Yaskawa INFORM job: R1_W03,5,7(0,0)OK-KM.JBI

/JOB
//NAME R1_W03,5,7(0,0)OK-KM
///FOLDERNAME KRIS-SCIANA
//POS
///NPOS 94,94,0,4,0,0
///TOOL 0
///POSTYPE PULSE
///PULSE
C00000=-97801,-92951,-68020,-42573,91743,12282
C00001=-188064,-59139,-49719,-51220,48350,5801
C00002=-182482,-29523,-13831,-58220,47542,10694
C00003=-186503,-14327,-833,-57181,45005,9773
C00004=-186887,-13436,-157,-57022,44797,9650
C00005=-187358,-18276,-5525,-56185,44980,9089
C00006=-193250,-27913,-6363,-58294,38967,9969
C00007=-199995,-16364,1412,-54222,35645,7165
C00008=-199327,-15584,1994,-54497,36056,7364
C00009=-199882,-17213,782,-54333,35681,7234
C00010=-195511,-15034,9725,-61255,35872,11434
C00011=-195511,-14418,11078,-61887,35615,11785
C00012=-194782,-15937,9357,-61766,36202,11793
C00013=-185148,-27392,-13403,-56780,46393,9588
C00014=-194611,-49573,-33459,-572,31924,22077
C00015=-195793,-42632,-27790,753,32004,21336
C00016=-196651,-38308,-23003,1749,31294,20781
C00017=-197052,-37261,-22343,2197,31434,20529
C00018=-196235,-39864,-25459,1248,31997,21059
C00019=-202582,-39238,-15691,30047,22851,6468
C00020=-202582,-38747,-14553,30589,22461,6206
C00021=-199520,-48265,-22642,26019,21519,8620
C00022=-195597,-45769,-34616,-8656,41829,26358
C00023=-205752,-37498,-18561,12983,36783,12907
C00024=-204602,-36516,-17940,11961,36728,13544
C00025=-195976,-39153,-18531,-9623,35365,26897
C00026=-197793,-59286,-35313,-7977,35152,25873
C00027=-213331,-48054,-41686,-15165,61809,-3623
C00028=-205738,-19523,-29471,-74829,71236,-32232
C00029=-213283,8162,-7439,-90948,66894,-41154
C00030=-215606,11272,-4686,-90700,65214,-41123
C00031=-216577,12559,-3127,-90719,64506,-40980
C00032=-216866,14771,-1122,-90727,64291,-40934
C00033=-216575,12516,-3571,-90601,64514,-41108
C00034=-216096,11995,12560,-96030,67022,-42309
C00035=-217024,11210,11856,-96058,66343,-42301
C00036=-218189,6682,-8739,-75138,67073,-44258
C00037=-217766,7327,-6835,-75554,67132,-43814
C00038=-218002,9228,-4372,-75728,66817,-43579
C00039=-221147,-8168,-21082,-78731,52920,-40929
C00040=-218126,-14316,-25848,-79593,55000,-40534
C00041=-213331,-48054,-41686,-15165,61809,-3623
C00042=-211970,-37779,-14430,-6801,34223,-17849
C00043=-210033,-36470,-13605,-8545,34568,-16753
C00044=-209079,-35786,-13170,-9389,34755,-16221
C00045=-208450,-36922,-14985,-9824,35355,-15936
C00046=-209854,-36909,-13406,-8784,34242,-16610
C00047=-205470,-32937,-11332,-12488,35564,-14251
C00048=-204626,-32211,-10856,-14325,36093,-12193
C00049=-199978,-27752,-7871,-22858,40221,2524
C00050=-194869,-21825,-3734,-26674,42807,10107
C00051=-213331,-48054,-41686,-15165,61809,-3623
C00052=-227702,13168,7438,-35164,58309,54158
C00053=-229907,15731,9772,-34304,57311,53471
C00054=-230826,16879,10578,-33881,57022,53136
C00055=-230146,17374,11284,-34234,57142,53417
C00056=-230917,15364,8500,-33669,57403,52958
C00057=-230398,6126,1186,-31847,60996,52995
C00058=-230715,5540,811,-31747,60817,52910
C00059=-229386,5021,240,-32222,61390,53323
C00060=-231429,-37745,-3451,-102210,21374,67263
C00061=-237321,-20462,7389,-96315,21390,64505
C00062=-234838,-16511,14692,-101345,23406,67189
C00063=-234421,-15866,15740,-101866,23741,67491
C00064=-232425,-13105,21006,-104766,25441,69160
C00065=-228509,-20375,12819,-100199,27869,67373
C00066=-227083,2935,-1542,-33047,62300,54059
C00067=-213331,-48054,-41686,-15165,61809,-3623
C00068=-211661,-57251,-25562,55725,28615,3338
C00069=-209733,-56166,-24995,54213,27635,4283
C00070=-230805,-7311,48072,113008,67410,-39116
C00071=-207937,-56864,-25063,53502,26430,4804
C00072=-210138,-56838,-26044,54013,28046,4347
C00073=-231104,-6899,48807,112946,67664,-39198
C00074=-231458,-6104,50179,112925,68017,-39364
C00075=-234772,6260,70319,113130,71928,-41806
C00076=-237075,19550,90913,113321,75131,-44224
C00077=-235689,-19373,32035,92744,56691,-36798
C00078=-221756,-61566,-27753,68083,36274,-1881
C00079=-225369,-69260,-37480,66382,39447,-1288
C00080=-205312,-39468,-16273,14091,10779,39550
C00081=-202035,-29821,-9269,1691,11105,45367
C00082=-201708,-29499,-9054,507,11133,45924
C00083=-224229,-15538,576,70048,44286,9521
C00084=-201579,-30109,-10785,40,11885,46143
C00085=-201147,-30171,-8613,-1607,10520,46916
C00086=-218609,-12576,2817,68837,40577,10645
C00087=-214363,-9679,5058,67669,37799,11594
C00088=-192443,-23943,-5231,-28759,13289,59765
C00089=-194260,-31922,-10655,-25195,12023,58034
C00090=-194296,-50223,-21768,-31420,9737,60851
C00091=-140544,-88669,-51716,-31420,85002,60851
C00092=-29274,49299,-4686,-19206,94492,76966
C00093=18103,108044,15339,-14006,98532,83827
BC00000=365145,1359,801155
BC00001=394627,15,902275
BC00002=366765,15,902279
BC00003=366765,15,902279
BC00004=366765,15,902279
BC00005=366765,15,902279
BC00006=366765,15,902279
BC00007=366765,15,902279
BC00008=366765,15,902279
BC00009=366765,15,902279
BC00010=366765,15,902279
BC00011=366765,15,902279
BC00012=366765,15,902279
BC00013=366765,15,902279
BC00014=338891,15,936852
BC00015=338891,15,936852
BC00016=338891,15,936852
BC00017=338891,15,936852
BC00018=338891,15,936852
BC00019=338891,15,936852
BC00020=338891,15,936852
BC00021=338891,15,936852
BC00022=338891,15,936852
BC00023=338891,15,936852
BC00024=338891,15,936852
BC00025=338891,15,936852
BC00026=338891,15,936852
BC00027=342850,15,986212
BC00028=385628,346,665290
BC00029=398174,443,571169
BC00030=398174,15,562195
BC00031=398174,15,558605
BC00032=398174,15,558605
BC00033=398174,15,558605
BC00034=398174,15,623710
BC00035=398174,15,623710
BC00036=398174,15,623710
BC00037=398174,15,623710
BC00038=398174,15,623710
BC00039=398174,15,575511
BC00040=398174,15,592196
BC00041=342850,15,986212
BC00042=339714,15,985872
BC00043=334030,15,972826
BC00044=331189,15,966303
BC00045=331189,15,966303
BC00046=331189,15,966303
BC00047=340653,15,937792
BC00048=341558,15,936829
BC00049=344452,15,937115
BC00050=349728,15,923193
BC00051=342850,15,986212
BC00052=398174,15,874824
BC00053=398174,15,860340
BC00054=398174,15,853098
BC00055=398174,15,853098
BC00056=398174,15,853098
BC00057=398174,15,815475
BC00058=398174,16,815473
BC00059=398174,15,823319
BC00060=398174,15,823316
BC00061=398175,16,823313
BC00062=398175,16,823313
BC00063=398175,16,823313
BC00064=398175,16,823313
BC00065=398175,16,823313
BC00066=398174,15,839006
BC00067=342850,15,986212
BC00068=326356,15,949986
BC00069=319697,15,940605
BC00070=317034,15,936852
BC00071=317034,15,936852
BC00072=317034,15,936852
BC00073=317034,15,936852
BC00074=317034,15,936852
BC00075=317034,15,936852
BC00076=317034,15,936852
BC00077=317034,15,936852
BC00078=317018,15,827734
BC00079=323550,15,836424
BC00080=372789,15,924496
BC00081=372967,15,918729
BC00082=365724,15,907858
BC00083=362827,15,903510
BC00084=362827,15,903510
BC00085=362827,15,903510
BC00086=362827,15,903510
BC00087=362827,15,903510
BC00088=365937,15,908086
BC00089=373180,15,918957
BC00090=373180,15,918957
BC00091=373180,15,918957
BC00092=212741,495,1019883
BC00093=144428,700,1062856
///POSTYPE BASE
///RECTAN
///RCONF 0,0,0,0,1,0,0,0,0,0,0,0,0,0,0,0,0,0,0,0,0,0,0,0
P00006=2.006,1.622,-0.565,0.0000,0.0000,0.0000
P00021=0.073,2.058,-0.109,0.0000,0.0000,0.0000
///RCONF 0,0,0,0,0,0,0,0,0,0,0,0,0,0,0,0,0,0,0,0,0,0,0,0
P00024=-1.466,-0.226,-0.419,0.0000,0.0000,0.0000
P00027=2.278,0.099,-4.210,0.0000,0.0000,0.0000
//INST
///DATE 2025/04/11 10:02
///ATTR SC,RW
///GROUP1 RB1,BS1
NOP
SFTOF
MOVJ C00000 BC00000 VJ=100.00
MOVJ C00001 BC00001 VJ=100.00
MOVJ C00002 BC00002 VJ=100.00
MOVL C00003 BC00003 V=60.0
REFP 3 C00004 BC00004
CALL JOB:SEARCH-R1
SET P021 P006
SFTON P021
MOVL C00005 BC00005 V=60.0
MOVL C00006 BC00006 V=100.0
MOVL C00007 BC00007 V=60.0
REFP 3 C00008 BC00008
CALL JOB:SEARCH-R1
SET P021 P006
SFTON P021
MOVL C00009 BC00009 V=60.0
MOVL C00010 BC00010 V=60.0
REFP 3 C00011 BC00011
CALL JOB:SEARCH-R1
SET P021 P006
SFTON P021
MOVL C00012 BC00012 V=60.0
MOVL C00013 BC00013 V=166.7
'Path S787 (for W405)
SFTOF
MOVL C00014 BC00014 V=100.0
MOVL C00015 BC00015 V=100.0
MOVL C00016 BC00016 V=60.0
REFP 3 C00017 BC00017
CALL JOB:SEARCH-R1
SET P027 P006
SFTON P027
MOVL C00018 BC00018 V=60.0
MOVL C00019 BC00019 V=60.0
REFP 3 C00020 BC00020
CALL JOB:SEARCH-R1
SET P027 P006
SFTON P027
MOVL C00021 BC00021 V=60.0
MOVL C00022 BC00022 V=100.0
MOVL C00023 BC00023 V=60.0
REFP 3 C00024 BC00024
CALL JOB:SEARCH-R1
SET P027 P006
SFTON P027
MOVL C00025 BC00025 V=60.0
MOVL C00026 BC00026 V=166.7
MOVJ C00027 BC00027 VJ=100.00
'Path S784 (for W404)
SFTOF
MOVJ C00028 BC00028 VJ=100.00
MOVJ C00029 BC00029 VJ=100.00
MOVJ C00030 BC00030 VJ=100.00
MOVL C00031 BC00031 V=100.0
REFP 3 C00032 BC00032
CALL JOB:SEARCH-R1
SET P024 P006
SFTON P024
MOVL C00033 BC00033 V=60.0
MOVL C00034 BC00034 V=60.0
REFP 3 C00035 BC00035
CALL JOB:SEARCH-R1
SET P024 P006
SFTON P024
MOVL C00036 BC00036 V=60.0
MOVL C00037 BC00037 V=60.0
REFP 3 C00038 BC00038
CALL JOB:SEARCH-R1
SET P024 P006
SFTON P024
MOVL C00039 BC00039 V=60.0
MOVL C00040 BC00040 V=166.7
MOVJ C00041 BC00041 VJ=100.00
'Path W402
SFTOF
CALL JOB:COFNIJ_DRUT
SFTON P021
MOVJ C00042 BC00042 VJ=100.00
MOVJ C00043 BC00043 VJ=100.00
MOVL C00044 BC00044 V=100.0 PL=0
REFP 1 C00045 BC00045
REFP 2 C00046 BC00046
MACRO1 MJ#(0) ARGF10
ARCON
MOVL C00047 BC00047 V=13.3
MOVL C00048 BC00048 V=13.3
MOVL C00049 BC00049 V=13.3
MOVL C00050 BC00050 V=13.3
ARCOF
SFTOF
'
MOVJ C00051 BC00051 VJ=100.00
'
'Path W866
SFTOF
SFTON P024
MOVL C00052 BC00052 V=166.7
MOVL C00053 BC00053 V=166.7
MOVL C00054 BC00054 V=100.0 PL=0
REFP 1 C00055 BC00055
REFP 2 C00056 BC00056
MACRO1 MJ#(0) ARGF10
ARCON
MOVL C00057 BC00057 V=13.3
MOVL C00058 BC00058 V=11.7
ARCOF
MOVL C00059 BC00059 V=166.7
MOVL C00060 BC00060 V=166.7
MACRO1 MJ#(0) ARGF7
MOVL C00061 BC00061 V=166.7
ARCON
MOVL C00062 BC00062 V=11.7
MOVL C00063 BC00063 V=11.7
MOVL C00064 BC00064 V=11.7
ARCOF
MOVL C00065 BC00065 V=166.7
MOVL C00066 BC00066 V=166.7
SFTOF
'
MOVJ C00067 BC00067 VJ=100.00
'
'Path W405
SFTOF
SFTON P027
MOVL C00068 BC00068 V=166.7
MOVL C00069 BC00069 V=166.7
MOVL C00070 BC00070 V=100.0 PL=0
REFP 1 C00071 BC00071
REFP 2 C00072 BC00072
MACRO1 MJ#(0) ARGF10
ARCON
MOVL C00073 BC00073 V=13.3
MOVL C00074 BC00074 V=13.3
MOVL C00075 BC00075 V=13.3
MOVL C00076 BC00076 V=13.3
MOVL C00077 BC00077 V=13.3
ARCOF
MOVL C00078 BC00078 V=166.7
MOVL C00079 BC00079 V=166.7
SFTOF
MOVJ C00080 BC00080 VJ=100.00
'Path W406
SFTOF
SFTON P027
MOVL C00081 BC00081 V=166.7
MOVL C00082 BC00082 V=166.7
MACRO1 MJ#(0) ARGF9
MOVL C00083 BC00083 V=100.0 PL=0
ARCON
REFP 1 C00084 BC00084
REFP 2 C00085 BC00085
MACRO1 MJ#(0) ARGF7
MOVL C00086 BC00086 V=10.8
MOVL C00087 BC00087 V=10.8
ARCOF
WVOF
MOVL C00088 BC00088 V=166.7
MOVL C00089 BC00089 V=166.7
SFTOF
MOVJ C00090 BC00090 VJ=100.00
MOVJ C00091 BC00091 VJ=100.00
MOVJ C00092 BC00092 VJ=100.00
MOVJ C00093 BC00093 VJ=100.00
END
